// SIMATIC S7-200 project (STEP 7-Micro/WIN), CPU 224 REL 02.01

ORGANIZATION_BLOCK MAIN:OB1
TITLE=PROGRAM COMMENTS
BEGIN
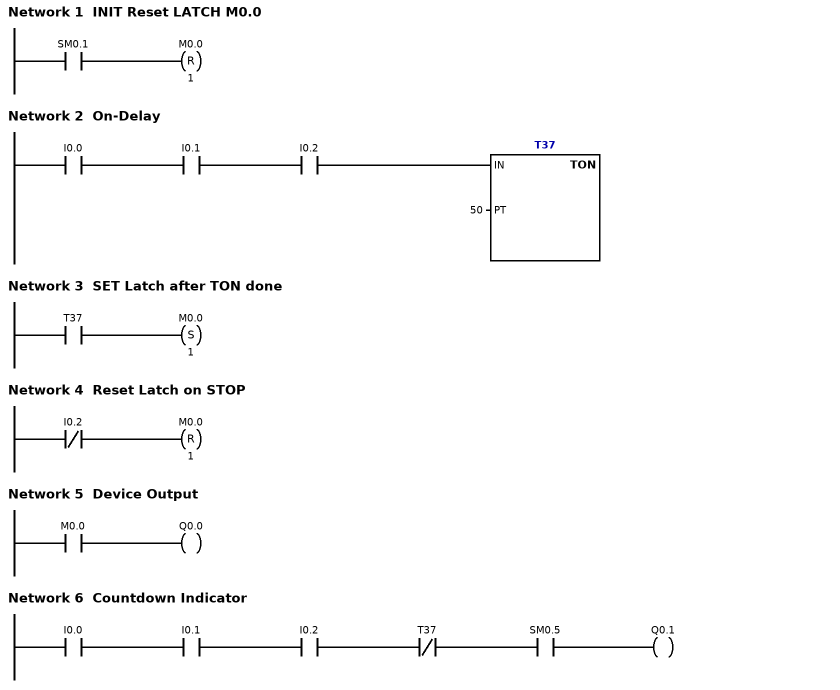
Network 1 // INIT Reset LATCH M0.0 
LD     SM0.1
R      M0.0, 1
Network 2 // On-Delay 
LD     I0.0
A      I0.1
A      I0.2
TON    T37, 50
Network 3 // SET Latch after TON done
LD     T37
S      M0.0, 1
Network 4 // Reset Latch on STOP
LDN    I0.2
R      M0.0, 1
Network 5 // Device Output
LD     M0.0
=      Q0.0
Network 6 // Countdown Indicator
LD     I0.0
A      I0.1
A      I0.2
AN     T37
A      SM0.5
=      Q0.1
END_ORGANIZATION_BLOCK
